Yaskawa INFORM job: R2_W53-A4(90,0)(Z_REKI)AWOK.JBI

/JOB
//NAME R2_W53-A4(90,0)(Z_REKI)AWOK
///FOLDERNAME AWOK
//POS
///NPOS 24,24,0,2,0,0
///TOOL 0
///POSTYPE PULSE
///PULSE
C00000=120458,47711,-19664,-12728,104208,-22558
C00001=120645,48979,-14537,-12631,101787,-22248
C00002=120718,49574,-12409,-12599,100816,-22125
C00003=120723,48768,-12014,-12567,100177,-22056
C00004=120718,49574,-12409,-12599,100816,-22125
C00005=120554,49259,-12918,-12560,100942,-22187
C00006=120558,50601,-11423,-12550,100718,-22162
C00007=120554,49259,-12918,-12560,100942,-22187
C00008=120639,49261,-12949,-12585,100973,-22166
C00009=121306,49268,-12942,-12775,101061,-21976
C00010=120639,49736,-12421,-12581,100894,-22157
C00011=120566,49145,-14546,-12613,101865,-22279
C00012=120377,47889,-19664,-12711,104287,-22590
C00013=118324,58007,-3629,-7223,91556,-33825
C00014=118324,55979,-2517,-7213,89843,-33726
C00015=118366,55063,-2566,-7228,89409,-33691
C00016=117769,53841,-3568,-7004,89352,-33862
C00017=118319,55966,-2495,-7211,89822,-33727
C00018=120938,57802,2770,-15654,86948,-24813
C00019=125029,61223,10317,-30462,86506,-23219
C00020=126996,60242,6149,-31134,88929,-23185
C00021=128970,69201,2441,-32101,95470,-24336
C00022=128973,76561,1055,-32522,99418,-25477
C00023=128973,76561,1055,-32522,99418,-25477
BC00000=269740,188520,1075175
BC00001=269740,188520,1075175
BC00002=269740,188520,1075175
BC00003=269740,188520,1075175
BC00004=269740,188520,1075175
BC00005=269740,188520,1075175
BC00006=269740,188520,1075175
BC00007=269740,188520,1075175
BC00008=269740,188520,1075175
BC00009=269740,188520,1075175
BC00010=269740,188520,1075175
BC00011=269740,188520,1075175
BC00012=269740,188520,1075175
BC00013=266395,221037,1075175
BC00014=265144,216294,1075175
BC00015=264781,214916,1075175
BC00016=264644,214396,1075175
BC00017=264644,214396,1075175
BC00018=264781,214916,1075175
BC00019=264781,214916,1075175
BC00020=264781,214916,1075175
BC00021=264781,214916,1075175
BC00022=264781,214916,1075175
BC00023=264781,527671,1075175
///POSTYPE BASE
///RECTAN
///RCONF 0,0,0,0,0,0,0,0,0,0,0,0,0,0,0,0,0,0,0,0,0,0,0,0
P00006=0.222,-3.123,-1.508,0.0000,0.0000,0.0000
P00024=0.145,-0.552,1.326,0.0000,0.0000,0.0000
//INST
///DATE 2023/11/01 17:02
///ATTR SC,RW
///GROUP1 RB1,BS1
NOP
'r2_W53-A4(90,0)(z_reki)
'Path S1026
SFTOF
MOVL C00000 BC00000 V=1000.0
MOVL C00001 BC00001 V=400.0
MOVL C00002 BC00002 V=60.0
REFP 3 C00003 BC00003
CALL JOB:SEARCH-R1
SET P024 P006
SFTON P024
MOVL C00004 BC00004 V=60.0
MOVL C00005 BC00005 V=60.0
REFP 3 C00006 BC00006
CALL JOB:SEARCH-R1
SET P024 P006
SFTON P024
MOVL C00007 BC00007 V=60.0
MOVL C00008 BC00008 V=60.0
REFP 3 C00009 BC00009
CALL JOB:SEARCH-R1
SET P024 P006
SFTON P024
MOVL C00010 BC00010 V=60.0
MOVL C00011 BC00011 V=400.0
MOVL C00012 BC00012 V=1000.0
'Path W1027
SFTOF
SFTON P024
MOVJ C00013 BC00013 VJ=100.00
MOVL C00014 BC00014 V=400.0
MOVL C00015 BC00015 V=100.0 PL=0
REFP 1 C00016 BC00016
REFP 2 C00017 BC00017
MACRO1 MJ#(0) ARGF9
ARCON
MOVL C00018 BC00018 V=10.8
MOVL C00019 BC00019 V=10.8
ARCOF
MOVL C00020 BC00020 V=400.0
MOVL C00021 BC00021 V=1000.0
SFTOF
'
MOVJ C00022 BC00022 VJ=50.00
MOVJ C00023 BC00023 VJ=50.00
END
